FUNCTION_BLOCK TFValutaAssiInFinestraDiPassMode
VAR_INPUT
	ModuleAX_X : POINTER TO TFModulePalletizer_Ax;
	ModuleAX_Y : POINTER TO TFModulePalletizer_Ax;
	ModuleAX_Z : POINTER TO TFModulePalletizer_Ax;
	ModuleAX_J : POINTER TO TFModulePalletizer_AxJ_Lastre;
	Traiettoria : POINTER TO TFTraiettoria;
	WorkAreaManager : POINTER TO TFWorkAreaManager;
END_VAR
VAR
	Direzione_X_Positiva : BOOL;
	Direzione_Y_Positiva : BOOL;
	Direzione_Z_Positiva : BOOL;
	Direzione_J_Positiva : BOOL;
	Direzione_K_Positiva : bool;
	AsseXInMoto: BOOL;
	AsseYInMoto: BOOL;
	AsseZInMoto: BOOL;
	AsseJInMoto: BOOL;
	//AsseKInMoto: BOOL;
	OffsetPassModeY_Appoggio: REAL;
END_VAR

(* Azzero le variabili *)
Asse_X_InFinestraDiPassMode := FALSE;
Asse_Y_InFinestraDiPassMode := FALSE;
Asse_Z_InFinestraDiPassMode := FALSE;
Asse_J_InFinestraDiPassMode := FALSE;

(* Valuto la direzione degli assi *)
Direzione_X_Positiva := TFDirezioneAssePositiva(Posizione_Attuale:=ModuleAX_X^.Ax^.Status.ActPosition,Posizione_Finale:=ProgrammaToModule_X.Quota_Destinazione);
Direzione_Y_Positiva := TFDirezioneAssePositiva(Posizione_Attuale:=ModuleAX_Y^.Ax^.Status.ActPosition,Posizione_Finale:=ProgrammaToModule_Y.Quota_Destinazione);
Direzione_Z_Positiva := TFDirezioneAssePositiva(Posizione_Attuale:=ModuleAX_Z^.Ax^.Status.ActPosition,Posizione_Finale:=ProgrammaToModule_Z.Quota_Destinazione);
Direzione_J_Positiva := TFDirezioneAssePositiva(Posizione_Attuale:=ModuleAX_J^.Ax^.Status.ActPosition,Posizione_Finale:=ProgrammaToModule_J.Quota_Destinazione);
(* Valuto se gli assi si stanno muovendo *)
AsseXInMoto:=ModuleAX_X^.Ax^.AxRef^.Status.Moving;
AsseYInMoto:=ModuleAX_Y^.Ax^.AxRef^.Status.Moving;
AsseZInMoto:=ModuleAX_Z^.Ax^.AxRef^.Status.Moving;
AsseJInMoto:=ModuleAX_J^.Ax^.AxRef^.Status.Moving;

IF Traiettoria^.PassModeGlobalEnable AND AbilitazionePassModeGlobale THEN (* Abilitazione Globale del PassMode*)
	
//	CASE WorkAreaManager^.State OF
		
//		WAMANAGER_CICLO_RIPOSO_RUN: 
			(* Abilito tutti i pasmode*)
			Traiettoria^.PassModePoint_X_Enable[1] := TRUE; 
			Traiettoria^.PassModePoint_Y_Enable[1] := TRUE; 
			Traiettoria^.PassModePoint_Z_Enable[1] := TRUE;
			Traiettoria^.PassModePoint_J_Enable[1] := TRUE;
			Traiettoria^.PassModePoint_K_Enable[1] := TRUE;
			(* Valuta il Pass Mode Per L'asse X *)
			IF Traiettoria^.PassModePoint_X_Enable[1] THEN
				IF AsseXInMoto THEN
					IF Direzione_X_Positiva THEN	//Se l'asse si sta muovendo in direzione POSITIVA
						IF ModuleAX_X^.Ax^.Status.ActPosition >= (ProgrammaToModule_X.Quota_Destinazione - OffsetPassMode.X) THEN
							Asse_X_InFinestraDiPassMode := TRUE;	
						END_IF
					ELSE							//Se l'asse si sta muovendo in direzione NEGATIVA
						IF ModuleAX_X^.Ax^.Status.ActPosition <= (ProgrammaToModule_X.Quota_Destinazione + OffsetPassMode.X) THEN
							Asse_X_InFinestraDiPassMode := TRUE;	
						END_IF
					END_IF
				END_IF
			END_IF
				
			(* Valuta il Pass Mode Per L'asse Y *)
			IF Traiettoria^.PassModePoint_Y_Enable[1] THEN
				IF Pinza_InIngombroColonne_Attuale THEN
					OffsetPassModeY_Appoggio := 80;
				ELSE
					OffsetPassModeY_Appoggio := OffsetPassMode.Y;
				END_IF
				IF AsseYInMoto THEN
					IF Direzione_Y_Positiva THEN	//Se l'asse si sta muovendo in direzione POSITIVA
						IF ModuleAX_Y^.Ax^.Status.ActPosition >= (ProgrammaToModule_Y.Quota_Destinazione - OffsetPassModeY_Appoggio) THEN
							Asse_Y_InFinestraDiPassMode := TRUE;	
						END_IF
					ELSE							//Se l'asse si sta muovendo in direzione NEGATIVA
						IF ModuleAX_Y^.Ax^.Status.ActPosition <= (ProgrammaToModule_Y.Quota_Destinazione + OffsetPassModeY_Appoggio) THEN
							Asse_Y_InFinestraDiPassMode := TRUE;	
						END_IF
					END_IF
				END_IF
			END_IF
			
			(* Valuta il Pass Mode Per L'asse Z *)
			IF Traiettoria^.PassModePoint_Z_Enable[1] THEN
				IF AsseZInMoto THEN
					IF Direzione_Z_Positiva THEN	//Se l'asse si sta muovendo in direzione POSITIVA
						IF ModuleAX_Z^.Ax^.Status.ActPosition >= (ProgrammaToModule_Z.Quota_Destinazione - OffsetPassMode.Z) THEN
							Asse_Z_InFinestraDiPassMode := TRUE;	
						END_IF
					ELSE							//Se l'asse si sta muovendo in direzione NEGATIVA
						IF ModuleAX_Z^.Ax^.Status.ActPosition <= (ProgrammaToModule_Z.Quota_Destinazione + OffsetPassMode.Z) THEN
							Asse_Z_InFinestraDiPassMode := TRUE;	
						END_IF
					END_IF
				END_IF
			END_IF
			
			(* Valuta il Pass Mode Per L'asse J *)
			IF Traiettoria^.PassModePoint_J_Enable[1] THEN
				IF AsseJInMoto THEN
					IF Direzione_J_Positiva THEN	//Se l'asse si sta muovendo in direzione POSITIVA
						IF ModuleAX_J^.Ax^.Status.ActPosition >= (ProgrammaToModule_J.Quota_Destinazione - OffsetPassMode.J) THEN
							Asse_J_InFinestraDiPassMode := TRUE;	
						END_IF
					ELSE							//Se l'asse si sta muovendo in direzione NEGATIVA
						IF ModuleAX_J^.Ax^.Status.ActPosition <= (ProgrammaToModule_J.Quota_Destinazione + OffsetPassMode.J) THEN
							Asse_J_InFinestraDiPassMode := TRUE;	
						END_IF
					END_IF
				END_IF
			END_IF
		(*
		WAMANAGER_CICLO_PRELIEVO_PALL_RUN: 
			(* Abilito tutti i pasmode*)
			Traiettoria^.PassModePoint_X_Enable[1] := TRUE; 
			Traiettoria^.PassModePoint_Y_Enable[1] := TRUE; 
			Traiettoria^.PassModePoint_Z_Enable[1] := TRUE;
			Traiettoria^.PassModePoint_J_Enable[1] := TRUE;
			Traiettoria^.PassModePoint_K_Enable[1] := TRUE;
			(* Valuta il Pass Mode Per L'asse X *)
			IF Traiettoria^.PassModePoint_X_Enable[1] THEN
				IF AsseXInMoto THEN
					IF Direzione_X_Positiva THEN	//Se l'asse si sta muovendo in direzione POSITIVA
						IF ModuleAX_X^.Ax^.Status.ActPosition >= (ProgrammaToModule_X.Quota_Destinazione - OffsetPassMode.X) THEN
							Asse_X_InFinestraDiPassMode := TRUE;	
						END_IF
					ELSE							//Se l'asse si sta muovendo in direzione NEGATIVA
						IF ModuleAX_X^.Ax^.Status.ActPosition <= (ProgrammaToModule_X.Quota_Destinazione + OffsetPassMode.X) THEN
							Asse_X_InFinestraDiPassMode := TRUE;	
						END_IF
					END_IF
				END_IF
			END_IF
				
			(* Valuta il Pass Mode Per L'asse Y *)
			IF Traiettoria^.PassModePoint_Y_Enable[1] THEN
				IF AsseYInMoto THEN
					IF Pinza_InIngombroColonne_Attuale THEN
						OffsetPassModeY_Appoggio := 80;
					ELSE
						OffsetPassModeY_Appoggio := OffsetPassMode.Y;
					END_IF
					IF Direzione_Y_Positiva THEN	//Se l'asse si sta muovendo in direzione POSITIVA
						IF ModuleAX_Y^.Ax^.Status.ActPosition >= (ProgrammaToModule_Y.Quota_Destinazione - OffsetPassModeY_Appoggio) THEN
							Asse_Y_InFinestraDiPassMode := TRUE;	
						END_IF
					ELSE							//Se l'asse si sta muovendo in direzione NEGATIVA
						IF ModuleAX_Y^.Ax^.Status.ActPosition <= (ProgrammaToModule_Y.Quota_Destinazione + OffsetPassModeY_Appoggio) THEN
							Asse_Y_InFinestraDiPassMode := TRUE;	
						END_IF
					END_IF	
				END_IF
			END_IF
			
			(* Valuta il Pass Mode Per L'asse Z *)
			IF Traiettoria^.PassModePoint_Z_Enable[1] THEN
				IF AsseZInMoto THEN
					IF Direzione_Z_Positiva THEN	//Se l'asse si sta muovendo in direzione POSITIVA
						IF ModuleAX_Z^.Ax^.Status.ActPosition >= (ProgrammaToModule_Z.Quota_Destinazione - OffsetPassMode.Z) THEN
							Asse_Z_InFinestraDiPassMode := TRUE;	
						END_IF
					ELSE							//Se l'asse si sta muovendo in direzione NEGATIVA
						IF ModuleAX_Z^.Ax^.Status.ActPosition <= (ProgrammaToModule_Z.Quota_Destinazione + OffsetPassMode.Z) THEN
							Asse_Z_InFinestraDiPassMode := TRUE;	
						END_IF
					END_IF
				END_IF
			END_IF
			
			(* Valuta il Pass Mode Per L'asse J *)
			IF Traiettoria^.PassModePoint_J_Enable[1] THEN
				IF AsseJInMoto THEN
					IF Direzione_J_Positiva THEN	//Se l'asse si sta muovendo in direzione POSITIVA
						IF ModuleAX_J^.Ax^.Status.ActPosition >= (ProgrammaToModule_J.Quota_Destinazione - OffsetPassMode.J) THEN
							Asse_J_InFinestraDiPassMode := TRUE;	
						END_IF
					ELSE							//Se l'asse si sta muovendo in direzione NEGATIVA
						IF ModuleAX_J^.Ax^.Status.ActPosition <= (ProgrammaToModule_J.Quota_Destinazione + OffsetPassMode.J) THEN
							Asse_J_InFinestraDiPassMode := TRUE;	
						END_IF
					END_IF
				END_IF
			END_IF
									
		WAMANAGER_CICLO_DEPOSITO_PALL_RUN: 
			(* Abilito tutti i pasmode*)
			Traiettoria^.PassModePoint_X_Enable[1] := TRUE; 
			Traiettoria^.PassModePoint_Y_Enable[1] := TRUE; 
			Traiettoria^.PassModePoint_Z_Enable[1] := TRUE;
			Traiettoria^.PassModePoint_J_Enable[1] := TRUE;
			Traiettoria^.PassModePoint_K_Enable[1] := TRUE;
			(* Valuta il Pass Mode Per L'asse X *)
			IF Traiettoria^.PassModePoint_X_Enable[1] THEN
				IF AsseXInMoto THEN
					IF Direzione_X_Positiva THEN	//Se l'asse si sta muovendo in direzione POSITIVA
						IF ModuleAX_X^.Ax^.Status.ActPosition >= (ProgrammaToModule_X.Quota_Destinazione - OffsetPassMode.X) THEN
							Asse_X_InFinestraDiPassMode := TRUE;	
						END_IF
					ELSE							//Se l'asse si sta muovendo in direzione NEGATIVA
						IF ModuleAX_X^.Ax^.Status.ActPosition <= (ProgrammaToModule_X.Quota_Destinazione + OffsetPassMode.X) THEN
							Asse_X_InFinestraDiPassMode := TRUE;	
						END_IF
					END_IF
				END_IF
			END_IF
				
			(* Valuta il Pass Mode Per L'asse Y *)
			IF Traiettoria^.PassModePoint_Y_Enable[1] THEN
				IF AsseYInMoto THEN
					IF Direzione_Y_Positiva THEN	//Se l'asse si sta muovendo in direzione POSITIVA
						IF ModuleAX_Y^.Ax^.Status.ActPosition >= (ProgrammaToModule_Y.Quota_Destinazione - OffsetPassMode.Y) THEN
							Asse_Y_InFinestraDiPassMode := TRUE;	
						END_IF
					ELSE							//Se l'asse si sta muovendo in direzione NEGATIVA
						IF ModuleAX_Y^.Ax^.Status.ActPosition <= (ProgrammaToModule_Y.Quota_Destinazione + OffsetPassMode.Y) THEN
							Asse_Y_InFinestraDiPassMode := TRUE;	
						END_IF
					END_IF
				END_IF
			END_IF
			
			(* Valuta il Pass Mode Per L'asse Z *)
			IF Traiettoria^.PassModePoint_Z_Enable[1] THEN
				IF AsseZInMoto THEN
					IF Direzione_Z_Positiva THEN	//Se l'asse si sta muovendo in direzione POSITIVA
						IF ModuleAX_Z^.Ax^.Status.ActPosition >= (ProgrammaToModule_Z.Quota_Destinazione - OffsetPassMode.Z) THEN
							Asse_Z_InFinestraDiPassMode := TRUE;	
						END_IF
					ELSE							//Se l'asse si sta muovendo in direzione NEGATIVA
						IF ModuleAX_Z^.Ax^.Status.ActPosition <= (ProgrammaToModule_Z.Quota_Destinazione + OffsetPassMode.Z) THEN
							Asse_Z_InFinestraDiPassMode := TRUE;	
						END_IF
					END_IF
				END_IF
			END_IF
			
			(* Valuta il Pass Mode Per L'asse J *)
			IF Traiettoria^.PassModePoint_J_Enable[1] THEN
				IF AsseJInMoto THEN
					IF Direzione_J_Positiva THEN	//Se l'asse si sta muovendo in direzione POSITIVA
						IF ModuleAX_J^.Ax^.Status.ActPosition >= (ProgrammaToModule_J.Quota_Destinazione - OffsetPassMode.J) THEN
							Asse_J_InFinestraDiPassMode := TRUE;	
						END_IF
					ELSE							//Se l'asse si sta muovendo in direzione NEGATIVA
						IF ModuleAX_J^.Ax^.Status.ActPosition <= (ProgrammaToModule_J.Quota_Destinazione + OffsetPassMode.J) THEN
							Asse_J_InFinestraDiPassMode := TRUE;	
						END_IF
					END_IF
				END_IF
			END_IF
									
		WAMANAGER_CICLO_PRELIEVO_FALDA_VUOTI_RUN:
			(* Abilito tutti i pasmode*)
			Traiettoria^.PassModePoint_X_Enable[1] := TRUE; 
			Traiettoria^.PassModePoint_Y_Enable[1] := TRUE; 
			Traiettoria^.PassModePoint_Z_Enable[1] := TRUE;
			Traiettoria^.PassModePoint_J_Enable[1] := TRUE;
			Traiettoria^.PassModePoint_K_Enable[1] := TRUE;
			(* Valuta il Pass Mode Per L'asse X *)
			IF Traiettoria^.PassModePoint_X_Enable[1] THEN
				IF AsseXInMoto THEN
					IF Direzione_X_Positiva THEN	//Se l'asse si sta muovendo in direzione POSITIVA
						IF ModuleAX_X^.Ax^.Status.ActPosition >= (ProgrammaToModule_X.Quota_Destinazione - OffsetPassMode.X) THEN
							Asse_X_InFinestraDiPassMode := TRUE;	
						END_IF
					ELSE							//Se l'asse si sta muovendo in direzione NEGATIVA
						IF ModuleAX_X^.Ax^.Status.ActPosition <= (ProgrammaToModule_X.Quota_Destinazione + OffsetPassMode.X) THEN
							Asse_X_InFinestraDiPassMode := TRUE;	
						END_IF
					END_IF
				END_IF
			END_IF
				
			(* Valuta il Pass Mode Per L'asse Y *)
			IF Traiettoria^.PassModePoint_Y_Enable[1] THEN
				IF Pinza_InIngombroColonne_Attuale THEN
					OffsetPassModeY_Appoggio := 80;
				ELSE
					OffsetPassModeY_Appoggio := OffsetPassMode.Y;
				END_IF
				IF AsseYInMoto THEN
					IF Direzione_Y_Positiva THEN	//Se l'asse si sta muovendo in direzione POSITIVA
						IF ModuleAX_Y^.Ax^.Status.ActPosition >= (ProgrammaToModule_Y.Quota_Destinazione - OffsetPassModeY_Appoggio) THEN
							Asse_Y_InFinestraDiPassMode := TRUE;	
						END_IF
					ELSE							//Se l'asse si sta muovendo in direzione NEGATIVA
						IF ModuleAX_Y^.Ax^.Status.ActPosition <= (ProgrammaToModule_Y.Quota_Destinazione + OffsetPassModeY_Appoggio) THEN
							Asse_Y_InFinestraDiPassMode := TRUE;	
						END_IF
					END_IF
				END_IF
			END_IF
			
			(* Valuta il Pass Mode Per L'asse Z *)
			IF Traiettoria^.PassModePoint_Z_Enable[1] THEN
				IF AsseZInMoto THEN
					IF Direzione_Z_Positiva THEN	//Se l'asse si sta muovendo in direzione POSITIVA
						IF ModuleAX_Z^.Ax^.Status.ActPosition >= (ProgrammaToModule_Z.Quota_Destinazione - OffsetPassMode.Z) THEN
							Asse_Z_InFinestraDiPassMode := TRUE;	
						END_IF
					ELSE							//Se l'asse si sta muovendo in direzione NEGATIVA
						IF ModuleAX_Z^.Ax^.Status.ActPosition <= (ProgrammaToModule_Z.Quota_Destinazione + OffsetPassMode.Z) THEN
							Asse_Z_InFinestraDiPassMode := TRUE;	
						END_IF
					END_IF
				END_IF
			END_IF
			
			(* Valuta il Pass Mode Per L'asse J *)
			IF Traiettoria^.PassModePoint_J_Enable[1] THEN
				IF AsseJInMoto THEN
					IF Direzione_J_Positiva THEN	//Se l'asse si sta muovendo in direzione POSITIVA
						IF ModuleAX_J^.Ax^.Status.ActPosition >= (ProgrammaToModule_J.Quota_Destinazione - OffsetPassMode.J) THEN
							Asse_J_InFinestraDiPassMode := TRUE;	
						END_IF
					ELSE							//Se l'asse si sta muovendo in direzione NEGATIVA
						IF ModuleAX_J^.Ax^.Status.ActPosition <= (ProgrammaToModule_J.Quota_Destinazione + OffsetPassMode.J) THEN
							Asse_J_InFinestraDiPassMode := TRUE;	
						END_IF
					END_IF
				END_IF
			END_IF
									
		WAMANAGER_CICLO_DEPOSITO_FALDA_VUOTI_RUN:
			(* Abilito tutti i pasmode*)
			Traiettoria^.PassModePoint_X_Enable[1] := TRUE; 
			Traiettoria^.PassModePoint_Y_Enable[1] := TRUE; 
			Traiettoria^.PassModePoint_Z_Enable[1] := TRUE;
			Traiettoria^.PassModePoint_J_Enable[1] := TRUE;
			Traiettoria^.PassModePoint_K_Enable[1] := TRUE;
			(* Valuta il Pass Mode Per L'asse X *)
			IF Traiettoria^.PassModePoint_X_Enable[1] THEN
				IF AsseXInMoto THEN
					IF Direzione_X_Positiva THEN	//Se l'asse si sta muovendo in direzione POSITIVA
						IF ModuleAX_X^.Ax^.Status.ActPosition >= (ProgrammaToModule_X.Quota_Destinazione - OffsetPassMode.X) THEN
							Asse_X_InFinestraDiPassMode := TRUE;	
						END_IF
					ELSE							//Se l'asse si sta muovendo in direzione NEGATIVA
						IF ModuleAX_X^.Ax^.Status.ActPosition <= (ProgrammaToModule_X.Quota_Destinazione + OffsetPassMode.X) THEN
							Asse_X_InFinestraDiPassMode := TRUE;	
						END_IF
					END_IF
				END_IF
			END_IF
				
			(* Valuta il Pass Mode Per L'asse Y *)
			IF Traiettoria^.PassModePoint_Y_Enable[1] THEN
				IF AsseYInMoto THEN
					IF Direzione_Y_Positiva THEN	//Se l'asse si sta muovendo in direzione POSITIVA
						IF ModuleAX_Y^.Ax^.Status.ActPosition >= (ProgrammaToModule_Y.Quota_Destinazione - OffsetPassMode.Y) THEN
							Asse_Y_InFinestraDiPassMode := TRUE;	
						END_IF
					ELSE							//Se l'asse si sta muovendo in direzione NEGATIVA
						IF ModuleAX_Y^.Ax^.Status.ActPosition <= (ProgrammaToModule_Y.Quota_Destinazione + OffsetPassMode.Y) THEN
							Asse_Y_InFinestraDiPassMode := TRUE;	
						END_IF
					END_IF
				END_IF
			END_IF
			
			(* Valuta il Pass Mode Per L'asse Z *)
			IF Traiettoria^.PassModePoint_Z_Enable[1] THEN
				IF AsseZInMoto THEN
					IF Direzione_Z_Positiva THEN	//Se l'asse si sta muovendo in direzione POSITIVA
						IF ModuleAX_Z^.Ax^.Status.ActPosition >= (ProgrammaToModule_Z.Quota_Destinazione - OffsetPassMode.Z) THEN
							Asse_Z_InFinestraDiPassMode := TRUE;	
						END_IF
					ELSE							//Se l'asse si sta muovendo in direzione NEGATIVA
						IF ModuleAX_Z^.Ax^.Status.ActPosition <= (ProgrammaToModule_Z.Quota_Destinazione + OffsetPassMode.Z) THEN
							Asse_Z_InFinestraDiPassMode := TRUE;	
						END_IF
					END_IF
				END_IF
			END_IF
			
			(* Valuta il Pass Mode Per L'asse J *)
			IF Traiettoria^.PassModePoint_J_Enable[1] THEN
				IF AsseJInMoto THEN
					IF Direzione_J_Positiva THEN	//Se l'asse si sta muovendo in direzione POSITIVA
						IF ModuleAX_J^.Ax^.Status.ActPosition >= (ProgrammaToModule_J.Quota_Destinazione - OffsetPassMode.J) THEN
							Asse_J_InFinestraDiPassMode := TRUE;	
						END_IF
					ELSE							//Se l'asse si sta muovendo in direzione NEGATIVA
						IF ModuleAX_J^.Ax^.Status.ActPosition <= (ProgrammaToModule_J.Quota_Destinazione + OffsetPassMode.J) THEN
							Asse_J_InFinestraDiPassMode := TRUE;	
						END_IF
					END_IF
				END_IF
			END_IF
		
		WAMANAGER_CICLO_PRELIEVO_FALDA_RUN:
			(* Abilito tutti i pasmode*)
			Traiettoria^.PassModePoint_X_Enable[1] := TRUE; 
			Traiettoria^.PassModePoint_Y_Enable[1] := TRUE; 
			Traiettoria^.PassModePoint_Z_Enable[1] := TRUE;
			Traiettoria^.PassModePoint_J_Enable[1] := TRUE;
			Traiettoria^.PassModePoint_K_Enable[1] := TRUE;
			(* Valuta il Pass Mode Per L'asse X *)
			IF Traiettoria^.PassModePoint_X_Enable[1] THEN
				IF AsseXInMoto THEN
					IF Direzione_X_Positiva THEN	//Se l'asse si sta muovendo in direzione POSITIVA
						IF ModuleAX_X^.Ax^.Status.ActPosition >= (ProgrammaToModule_X.Quota_Destinazione - OffsetPassMode.X) THEN
							Asse_X_InFinestraDiPassMode := TRUE;	
						END_IF
					ELSE							//Se l'asse si sta muovendo in direzione NEGATIVA
						IF ModuleAX_X^.Ax^.Status.ActPosition <= (ProgrammaToModule_X.Quota_Destinazione + OffsetPassMode.X) THEN
							Asse_X_InFinestraDiPassMode := TRUE;	
						END_IF
					END_IF
				END_IF
			END_IF
				
			(* Valuta il Pass Mode Per L'asse Y *)
			IF Traiettoria^.PassModePoint_Y_Enable[1] THEN
				IF Pinza_InIngombroColonne_Attuale THEN
					OffsetPassModeY_Appoggio := 80;
				ELSE
					OffsetPassModeY_Appoggio := OffsetPassMode.Y;
				END_IF
				IF AsseYInMoto THEN
					IF Direzione_Y_Positiva THEN	//Se l'asse si sta muovendo in direzione POSITIVA
						IF ModuleAX_Y^.Ax^.Status.ActPosition >= (ProgrammaToModule_Y.Quota_Destinazione - OffsetPassModeY_Appoggio) THEN
							Asse_Y_InFinestraDiPassMode := TRUE;	
						END_IF
					ELSE							//Se l'asse si sta muovendo in direzione NEGATIVA
						IF ModuleAX_Y^.Ax^.Status.ActPosition <= (ProgrammaToModule_Y.Quota_Destinazione + OffsetPassModeY_Appoggio) THEN
							Asse_Y_InFinestraDiPassMode := TRUE;	
						END_IF
					END_IF
				END_IF
			END_IF
			
			(* Valuta il Pass Mode Per L'asse Z *)
			IF Traiettoria^.PassModePoint_Z_Enable[1] THEN
				IF AsseZInMoto THEN
					IF Direzione_Z_Positiva THEN	//Se l'asse si sta muovendo in direzione POSITIVA
						IF ModuleAX_Z^.Ax^.Status.ActPosition >= (ProgrammaToModule_Z.Quota_Destinazione - OffsetPassMode.Z) THEN
							Asse_Z_InFinestraDiPassMode := TRUE;	
						END_IF
					ELSE							//Se l'asse si sta muovendo in direzione NEGATIVA
						IF ModuleAX_Z^.Ax^.Status.ActPosition <= (ProgrammaToModule_Z.Quota_Destinazione + OffsetPassMode.Z) THEN
							Asse_Z_InFinestraDiPassMode := TRUE;	
						END_IF
					END_IF
				END_IF
			END_IF
			
			(* Valuta il Pass Mode Per L'asse J *)
			IF Traiettoria^.PassModePoint_J_Enable[1] THEN
				IF AsseJInMoto THEN
					IF Direzione_J_Positiva THEN	//Se l'asse si sta muovendo in direzione POSITIVA
						IF ModuleAX_J^.Ax^.Status.ActPosition >= (ProgrammaToModule_J.Quota_Destinazione - OffsetPassMode.J) THEN
							Asse_J_InFinestraDiPassMode := TRUE;	
						END_IF
					ELSE							//Se l'asse si sta muovendo in direzione NEGATIVA
						IF ModuleAX_J^.Ax^.Status.ActPosition <= (ProgrammaToModule_J.Quota_Destinazione + OffsetPassMode.J) THEN
							Asse_J_InFinestraDiPassMode := TRUE;	
						END_IF
					END_IF
				END_IF
			END_IF
			
		WAMANAGER_CICLO_DEPOSITO_FALDA_RUN:
			(* Abilito tutti i pasmode*)
			Traiettoria^.PassModePoint_X_Enable[1] := TRUE; 
			Traiettoria^.PassModePoint_Y_Enable[1] := TRUE; 
			Traiettoria^.PassModePoint_Z_Enable[1] := TRUE;
			Traiettoria^.PassModePoint_J_Enable[1] := TRUE;
			Traiettoria^.PassModePoint_K_Enable[1] := TRUE;
			(* Valuta il Pass Mode Per L'asse X *)
			IF Traiettoria^.PassModePoint_X_Enable[1] THEN
				IF AsseXInMoto THEN
					IF Direzione_X_Positiva THEN	//Se l'asse si sta muovendo in direzione POSITIVA
						IF ModuleAX_X^.Ax^.Status.ActPosition >= (ProgrammaToModule_X.Quota_Destinazione - OffsetPassMode.X) THEN
							Asse_X_InFinestraDiPassMode := TRUE;	
						END_IF
					ELSE							//Se l'asse si sta muovendo in direzione NEGATIVA
						IF ModuleAX_X^.Ax^.Status.ActPosition <= (ProgrammaToModule_X.Quota_Destinazione + OffsetPassMode.X) THEN
							Asse_X_InFinestraDiPassMode := TRUE;	
						END_IF
					END_IF
				END_IF
			END_IF
				
			(* Valuta il Pass Mode Per L'asse Y *)
			IF Traiettoria^.PassModePoint_Y_Enable[1] THEN
				IF AsseYInMoto THEN
					IF Direzione_Y_Positiva THEN	//Se l'asse si sta muovendo in direzione POSITIVA
						IF ModuleAX_Y^.Ax^.Status.ActPosition >= (ProgrammaToModule_Y.Quota_Destinazione - OffsetPassMode.Y) THEN
							Asse_Y_InFinestraDiPassMode := TRUE;	
						END_IF
					ELSE							//Se l'asse si sta muovendo in direzione NEGATIVA
						IF ModuleAX_Y^.Ax^.Status.ActPosition <= (ProgrammaToModule_Y.Quota_Destinazione + OffsetPassMode.Y) THEN
							Asse_Y_InFinestraDiPassMode := TRUE;	
						END_IF
					END_IF
				END_IF
			END_IF
			
			(* Valuta il Pass Mode Per L'asse Z *)
			IF Traiettoria^.PassModePoint_Z_Enable[1] THEN
				IF AsseZInMoto THEN
					IF Direzione_Z_Positiva THEN	//Se l'asse si sta muovendo in direzione POSITIVA
						IF ModuleAX_Z^.Ax^.Status.ActPosition >= (ProgrammaToModule_Z.Quota_Destinazione - OffsetPassMode.Z) THEN
							Asse_Z_InFinestraDiPassMode := TRUE;	
						END_IF
					ELSE							//Se l'asse si sta muovendo in direzione NEGATIVA
						IF ModuleAX_Z^.Ax^.Status.ActPosition <= (ProgrammaToModule_Z.Quota_Destinazione + OffsetPassMode.Z) THEN
							Asse_Z_InFinestraDiPassMode := TRUE;	
						END_IF
					END_IF
				END_IF
			END_IF
			
			(* Valuta il Pass Mode Per L'asse J *)
			IF Traiettoria^.PassModePoint_J_Enable[1] THEN
				IF AsseJInMoto THEN
					IF Direzione_J_Positiva THEN	//Se l'asse si sta muovendo in direzione POSITIVA
						IF ModuleAX_J^.Ax^.Status.ActPosition >= (ProgrammaToModule_J.Quota_Destinazione - OffsetPassMode.J) THEN
							Asse_J_InFinestraDiPassMode := TRUE;	
						END_IF
					ELSE							//Se l'asse si sta muovendo in direzione NEGATIVA
						IF ModuleAX_J^.Ax^.Status.ActPosition <= (ProgrammaToModule_J.Quota_Destinazione + OffsetPassMode.J) THEN
							Asse_J_InFinestraDiPassMode := TRUE;	
						END_IF
					END_IF
				END_IF
			END_IF
		(*
		WAMANAGER_CICLO_PRELIEVO_PACCO_RUN:
			(* Abilito tutti i pasmode*)
			Traiettoria^.PassModePoint_X_Enable[1] := TRUE; 
			Traiettoria^.PassModePoint_Y_Enable[1] := TRUE; 
			Traiettoria^.PassModePoint_Z_Enable[1] := TRUE;
			Traiettoria^.PassModePoint_J_Enable[1] := TRUE;
			Traiettoria^.PassModePoint_K_Enable[1] := TRUE;
			(* Valuta il Pass Mode Per L'asse X *)
			IF Traiettoria^.PassModePoint_X_Enable[1] THEN
				IF AsseXInMoto THEN
					IF Direzione_X_Positiva THEN	//Se l'asse si sta muovendo in direzione POSITIVA
						IF ModuleAX_X^.Ax^.Status.ActPosition >= (ProgrammaToModule_X.Quota_Destinazione - OffsetPassMode.X) THEN
							Asse_X_InFinestraDiPassMode := TRUE;	
						END_IF
					ELSE							//Se l'asse si sta muovendo in direzione NEGATIVA
						IF ModuleAX_X^.Ax^.Status.ActPosition <= (ProgrammaToModule_X.Quota_Destinazione + OffsetPassMode.X) THEN
							Asse_X_InFinestraDiPassMode := TRUE;	
						END_IF
					END_IF
				END_IF
			END_IF
				
			(* Valuta il Pass Mode Per L'asse Y *)
			IF Traiettoria^.PassModePoint_Y_Enable[1] THEN
				IF Pinza_InIngombroColonne_Attuale THEN
					OffsetPassModeY_Appoggio := 80;
				ELSE
					OffsetPassModeY_Appoggio := OffsetPassMode.Y;
				END_IF
				IF AsseYInMoto THEN
					IF Direzione_Y_Positiva THEN	//Se l'asse si sta muovendo in direzione POSITIVA
						IF ModuleAX_Y^.Ax^.Status.ActPosition >= (ProgrammaToModule_Y.Quota_Destinazione - OffsetPassModeY_Appoggio) THEN
							Asse_Y_InFinestraDiPassMode := TRUE;	
						END_IF
					ELSE							//Se l'asse si sta muovendo in direzione NEGATIVA
						IF ModuleAX_Y^.Ax^.Status.ActPosition <= (ProgrammaToModule_Y.Quota_Destinazione + OffsetPassModeY_Appoggio) THEN
							Asse_Y_InFinestraDiPassMode := TRUE;	
						END_IF
					END_IF
				END_IF
			END_IF
			
			(* Valuta il Pass Mode Per L'asse Z *)
			IF Traiettoria^.PassModePoint_Z_Enable[1] THEN
				IF AsseZInMoto THEN
					IF Direzione_Z_Positiva THEN	//Se l'asse si sta muovendo in direzione POSITIVA
						IF ModuleAX_Z^.Ax^.Status.ActPosition >= (ProgrammaToModule_Z.Quota_Destinazione - OffsetPassMode.Z) THEN
							Asse_Z_InFinestraDiPassMode := TRUE;	
						END_IF
					ELSE							//Se l'asse si sta muovendo in direzione NEGATIVA
						IF ModuleAX_Z^.Ax^.Status.ActPosition <= (ProgrammaToModule_Z.Quota_Destinazione + OffsetPassMode.Z) THEN
							Asse_Z_InFinestraDiPassMode := TRUE;	
						END_IF
					END_IF
				END_IF
			END_IF
			
			(* Valuta il Pass Mode Per L'asse J *)
			IF Traiettoria^.PassModePoint_J_Enable[1] THEN
				IF AsseJInMoto THEN
					IF Direzione_J_Positiva THEN	//Se l'asse si sta muovendo in direzione POSITIVA
						IF ModuleAX_J^.Ax^.Status.ActPosition >= (ProgrammaToModule_J.Quota_Destinazione - 2(*OffsetPassMode.J*)) THEN
							Asse_J_InFinestraDiPassMode := TRUE;	
						END_IF
					ELSE							//Se l'asse si sta muovendo in direzione NEGATIVA
						IF ModuleAX_J^.Ax^.Status.ActPosition <= (ProgrammaToModule_J.Quota_Destinazione + 2(*OffsetPassMode.J*)) THEN
							Asse_J_InFinestraDiPassMode := TRUE;	
						END_IF
					END_IF
				END_IF
			END_IF
									
		WAMANAGER_CICLO_DEPOSITO_PACCO_RUN:
			(* Abilito tutti i pasmode*)
			Traiettoria^.PassModePoint_X_Enable[1] := TRUE; 
			Traiettoria^.PassModePoint_Y_Enable[1] := TRUE; 
			Traiettoria^.PassModePoint_Z_Enable[1] := TRUE;
			Traiettoria^.PassModePoint_J_Enable[1] := TRUE;
			Traiettoria^.PassModePoint_K_Enable[1] := TRUE;
			(* Valuta il Pass Mode Per L'asse X *)
			IF Traiettoria^.PassModePoint_X_Enable[1] THEN
				IF AsseXInMoto THEN
					IF Direzione_X_Positiva THEN	//Se l'asse si sta muovendo in direzione POSITIVA
						IF ModuleAX_X^.Ax^.Status.ActPosition >= (ProgrammaToModule_X.Quota_Destinazione - OffsetPassMode.X) THEN
							Asse_X_InFinestraDiPassMode := TRUE;	
						END_IF
					ELSE							//Se l'asse si sta muovendo in direzione NEGATIVA
						IF ModuleAX_X^.Ax^.Status.ActPosition <= (ProgrammaToModule_X.Quota_Destinazione + OffsetPassMode.X) THEN
							Asse_X_InFinestraDiPassMode := TRUE;	
						END_IF
					END_IF
				END_IF
			END_IF
				
			(* Valuta il Pass Mode Per L'asse Y *)
			IF Traiettoria^.PassModePoint_Y_Enable[1] THEN
				IF AsseYInMoto THEN
					IF Direzione_Y_Positiva THEN	//Se l'asse si sta muovendo in direzione POSITIVA
						IF ModuleAX_Y^.Ax^.Status.ActPosition >= (ProgrammaToModule_Y.Quota_Destinazione - OffsetPassMode.Y) THEN
							Asse_Y_InFinestraDiPassMode := TRUE;	
						END_IF
					ELSE							//Se l'asse si sta muovendo in direzione NEGATIVA
						IF ModuleAX_Y^.Ax^.Status.ActPosition <= (ProgrammaToModule_Y.Quota_Destinazione + OffsetPassMode.Y) THEN
							Asse_Y_InFinestraDiPassMode := TRUE;	
						END_IF
					END_IF
				END_IF
			END_IF
			
			(* Valuta il Pass Mode Per L'asse Z *)
			IF Traiettoria^.PassModePoint_Z_Enable[1] THEN
				IF AsseZInMoto THEN
					IF Direzione_Z_Positiva THEN	//Se l'asse si sta muovendo in direzione POSITIVA
						IF ModuleAX_Z^.Ax^.Status.ActPosition >= (ProgrammaToModule_Z.Quota_Destinazione - OffsetPassMode.Z) THEN
							Asse_Z_InFinestraDiPassMode := TRUE;	
						END_IF
					ELSE							//Se l'asse si sta muovendo in direzione NEGATIVA
						IF ModuleAX_Z^.Ax^.Status.ActPosition <= (ProgrammaToModule_Z.Quota_Destinazione + OffsetPassMode.Z) THEN
							Asse_Z_InFinestraDiPassMode := TRUE;	
						END_IF
					END_IF
				END_IF
			END_IF
			
			(* Valuta il Pass Mode Per L'asse J *)
			IF Traiettoria^.PassModePoint_J_Enable[1] THEN
				IF AsseJInMoto THEN
					IF Direzione_J_Positiva THEN	//Se l'asse si sta muovendo in direzione POSITIVA
						IF ModuleAX_J^.Ax^.Status.ActPosition >= (ProgrammaToModule_J.Quota_Destinazione - OffsetPassMode.J) THEN
							Asse_J_InFinestraDiPassMode := TRUE;	
						END_IF
					ELSE							//Se l'asse si sta muovendo in direzione NEGATIVA
						IF ModuleAX_J^.Ax^.Status.ActPosition <= (ProgrammaToModule_J.Quota_Destinazione + OffsetPassMode.J) THEN
							Asse_J_InFinestraDiPassMode := TRUE;	
						END_IF
					END_IF
				END_IF
			END_IF
	*)
	END_CASE*)


ELSE
	(* Disabilito tutti i PasMode*)
	Traiettoria^.PassModePoint_X_Enable[1] := FALSE; 
	Traiettoria^.PassModePoint_Y_Enable[1] := FALSE; 
	Traiettoria^.PassModePoint_Z_Enable[1] := FALSE;
	Traiettoria^.PassModePoint_J_Enable[1] := FALSE;
	Traiettoria^.PassModePoint_K_Enable[1] := FALSE;
END_IF

END_FUNCTION_BLOCK

(* stored: Version 1.1.0.1, ProductVersion 3.1.4024.11
   POU TFValutaAssiInFinestraDiPassMode: Id {8691e484-8401-4b68-83cf-b34a747e6c46}, SpecialFunc None *)
